FUNCTION_BLOCK FB_Sensor
VAR
	bInput		AT %I*	: BOOL;
	nInput		AT %I*	: BOOL;
	
END_VAR

END_FUNCTION_BLOCK

(* stored: Version 1.1.0.1, ProductVersion 3.1.4024.12
   POU FB_Sensor: Id {b88aef50-2f22-415c-b94d-4de550809054}, SpecialFunc None *)
